(*	1. New version of FB: FB_IPRO_ModbusRTU 
	2. I haven't test it yet.
*) 
FUNCTION_BLOCK FB_IproV2 EXTENDS FB_UniversalAxis IMPLEMENTS I_UniversalAxis, I_AxisMoveAbsolute
VAR
	eSystemStatus : E_IProStatus; 							(* r0.30 *)
	uPositionCmd : U_Word2Dint;
END_VAR

bError := bModbusError OR iErrorID<>0;
CASE eAxisState OF
	AXIS_INITIALIZING..AXIS_RESET_DONE, AXIS_ABORTING:
		tonConfirmReallyError(
			IN := bError OR bModbusError,
			PT := timeConfirmReallyError,
			Q => bReallyError 
		);
END_CASE
SUPER^();

(* Copy it to derived Function block if developing this function *)
PROPERTY ActualPosition : REFERENCE TO LREAL
GET
ActualPosition REF= lrActualPosition;
END_GET
END_PROPERTY

METHOD Convert : BOOL
VAR_INPUT
	iRegionNo	:	INT;
	pReadData	:	POINTER TO word;
END_VAR
VAR
	TempData	:	 U_Word2Dint;
END_VAR
TempData.iWord[0] := pReadData[0];
TempData.iWord[1] := pReadData[1];
CASE iRegionNo OF
	0:// position unit 1
		lrActualPosition := DINT_TO_LREAL(TempData.idInt); //64 bit
	1:// status read
		eSystemStatus := pReadData[0];
	2:// fault code
		iErrorID := pReadData[0];// must not use word to int
END_CASE
END_METHOD

(* Copy it to derived Function block if developing this function *)
PROPERTY InPosition : BOOL
GET
InPosition := F_CheckInRange( lrHighLimit := lrActualPosition+50,
						lrLowLimit := lrActualPosition-50,
						lrValue := lrAbsolutePosition);
END_GET
END_PROPERTY

METHOD MR_MoveAbsolute : BOOL
VAR_INPUT
	lrAbsolutePosition : LREAL;
END_VAR
IF eAxisState = AXIS_IDLE AND
	NOT F_InRange(
		bound1 := THIS^.lrAbsolutePosition + 50,
		bound2 := THIS^.lrAbsolutePosition - 50,
		value := lrAbsolutePosition,
	)
THEN
	THIS^.lrAbsolutePosition := lrAbsolutePosition;
	bMoveAbsolute := TRUE;
	bInPostion 	:= FALSE;
	bInVelocity := FALSE;
	bMoveActive := TRUE;
	bStopped 	:= FALSE;
	bHalted 	:= FALSE;
	bJogDone 	:= FALSE;
	
	eAxisState := AXIS_MOVE_ABSOLUTE;
	fbMachineLogger.MR_AddLogs(CONCAT(sName,' : move absolute requested'));		
	
ELSIF eAxisState = AXIS_MOVE_ABSOLUTE_DONE THEN
	bInPostion 		:= TRUE;
	bInVelocity		:= FALSE;
	bMoveActive 	:= FALSE;
	bStopped 		:= FALSE;
	bHalted			:= FALSE;
	bJogDone 		:= FALSE;
	bMoveAbsolute 	:= FALSE;
	MR_MoveAbsolute := TRUE;
	fbMachineLogger.MR_AddLogs(CONCAT(sName,' : move absolute done'));		
	
END_IF
END_METHOD

METHOD PROTECTED MS_Aborting
VAR_INPUT
END_VAR
arrAddressWrite[0][2] := 0;//disable servo
lrAbsolutePosition := 0;
eSystemStatus := IPRO_STATUS_NOT_RESPOND;	// reset status
eAxisState := AXIS_UNINITIALIZED;
END_METHOD

METHOD PROTECTED MS_Initializing
VAR_INPUT
END_VAR
SUPER^.MS_Initializing();
arrAddressWrite[0][2] := 1;	// enable Servo
 
IF eSystemStatus = IPRO_STATUS_RUN THEN
	eAxisState := AXIS_READY_INITIALIZED;
END_IF
END_METHOD

METHOD PROTECTED  MS_MoveAbsolute
VAR_INPUT
END_VAR
uPositionCmd.idInt := LREAL_TO_DINT(lrAbsolutePosition);
arrAddressWrite[1][2] := uPositionCmd.iWord[0];
arrAddressWrite[1][3] := uPositionCmd.iWord[1];

IF F_CheckInRange(lrHighLimit := lrAbsolutePosition + 50,
					lrLowLimit := lrAbsolutePosition - 50,
					lrValue := lrActualPosition)
THEN
	eAxisState := AXIS_MOVE_ABSOLUTE_DONE;
END_IF
END_METHOD

(* I havn't find the way to reset this servo yet *)
METHOD PROTECTED MS_Reset
VAR_INPUT
END_VAR
END_METHOD

METHOD PROTECTED MS_Uninitalized
VAR_INPUT
END_VAR
SUPER^.MS_Uninitalized();
bBusy := FALSE;
// Read
	arrAddressRead[0][0] := 4004;// motor position FB// reference unit 
	arrAddressRead[0][1] := 4;
	arrAddressRead[0][2] := E_ModbusFunction.ReadHoldingRegisters;
	
	arrAddressRead[1][0] := 4064;// System status // 
	arrAddressRead[1][1] := 1;
	arrAddressRead[1][2] := E_ModbusFunction.ReadHoldingRegisters;
	
	arrAddressRead[2][0] := 4198;// FaultCode
	arrAddressRead[2][1] := 1;
	arrAddressRead[2][2] := E_ModbusFunction.ReadHoldingRegisters;	
	
	iNumAddRegionRead := 3;
	
// write	
	arrAddressWrite[0][0] := 1822;//	enable servo 
	arrAddressWrite[0][1] := 1;
	arrAddressWrite[0][2] := 0; // 0: disable,  1: enable
	arrAddressWrite[0][10] := E_ModbusFunction.WriteSingleRegister;
	
	arrAddressWrite[1][0] := 1824;// 32 bit 1825
	arrAddressWrite[1][1] := 2;
	arrAddressWrite[1][2] := 0;
	arrAddressWrite[1][3] := 0;
	arrAddressWrite[1][10] := E_ModbusFunction.WriteMultipleRegisters;
	
	iNumAddRegionWrite := 2;
END_METHOD

(*Please note this properties currently return the lrAbsolutePosition,
-If you expand the FB to implement other I_AxisMove..., you need to change this property's implement, and this note.
*)
PROPERTY SetpointPosition : LREAL
GET
SetpointPosition := lrAbsolutePosition;
END_GET
END_PROPERTY

END_FUNCTION_BLOCK

(* stored: Version 1.1.0.1, ProductVersion 3.1.4024.12
   POU FB_IproV2: Id {a1850c55-91c3-4ab1-8e24-07ab3cc237b8}, SpecialFunc None
   Property ActualPosition: Id {c23867ff-70a6-4d76-92c5-d92c7b1f769f}
   Get Get: Id {c1768b23-7cc6-4fb8-8725-9787679389e4}
   Method Convert: Id {5c6c2c58-3d39-4e1a-927c-75d7424dced3}
   Property InPosition: Id {d37f148b-ff3f-4e48-b0e2-90024f1d89f6}
   Get Get: Id {95d56889-6b61-40f3-8cb9-8e7e54d31a8c}
   Method MR_MoveAbsolute: Id {50001668-ff58-4ca3-b81c-7b7f114d6d59}
   Method MS_Aborting: Id {2eb55b58-07b5-4a48-9783-5d0deaa34c78}
   Method MS_Initializing: Id {87bcaad7-643e-4f02-8293-980cd1078ebb}
   Method MS_MoveAbsolute: Id {d67e44d3-8c54-4147-bfc4-e9ff09ead217}
   Method MS_Reset: Id {d99a8526-91bf-41e7-8ca0-cd1b6fc70a52}
   Method MS_Uninitalized: Id {a41a3315-bf2d-4973-8d0f-2b1991284521}
   Property SetpointPosition: Id {3a238ae6-ab74-4aa3-a39d-5ab0a033ab2e}
   Get Get: Id {f66ef654-f874-4ecc-8330-83f0653d361a} *)
